{attribute 'enable_dynamic_creation'}
FUNCTION_BLOCK Cylinder_ExtendCommand EXTENDS AsynchronousCommand
VAR
	cylinder : I_Cylinder;
END_VAR

METHOD FB_init : BOOL
VAR_INPUT
	bInitRetains : BOOL; // if TRUE, the retain variables are initialized (warm start / cold start)
	bInCopyCode : BOOL;  // if TRUE, the instance afterwards gets moved into the copy code (online change)	
	Cylinder : I_Cylinder;
END_VAR
THIS^.cylinder := Cylinder;
END_METHOD

METHOD PROTECTED WhileBusy
VAR_INPUT
	commandState : I_AsynchronousCommandBusyState;
END_VAR
cylinder.FullyExtend();

IF cylinder.IsFullyExtended THEN
	commandState.SetDone();	
END_IF
END_METHOD

END_FUNCTION_BLOCK

(* stored: Version 1.1.0.1, ProductVersion 3.1.4024.11
   POU Cylinder_ExtendCommand: Id {7001d6b3-390f-4bb7-869a-6f280916d893}, SpecialFunc None
   Folder Constructor: Id {cfbe9121-ba24-4ee0-83c6-35c732c66db7}
   Folder Protected: Id {8238ea7e-58a5-40ba-8ada-21ad7be82f02}
   Method FB_init: Id {fd210eca-3d28-4f93-9854-14401eb2a1d7}
   Method WhileBusy: Id {5199f700-58c0-4dd7-8d14-13281507ed21} *)
